FUNCTION GetRevision : UINT
VAR_INPUT
END_VAR
VAR
END_VAR

GetRevision := Version.Revision;

END_FUNCTION

(* stored: Version 1.1.0.1, ProductVersion 3.1.4024.0
   POU GetRevision: Id {eb6328b5-aa83-432b-bb0a-272935f2df1a}, SpecialFunc None *)
